PROGRAM SC_MAIN_FSM
VAR
	main_fsm	: FB_Main_FSM;
	
END_VAR

main_fsm(currentCmd := GVL_FSM.E_CommandGlobal, EmergencyReason := GVL_FSM.E_EmergencyReasonGlobal);

END_PROGRAM

(* stored: Version 1.1.0.1
   POU SC_MAIN_FSM: Id {8ae7d21a-5b8b-4fb0-8d34-ff7e9a16183c}, SpecialFunc None *)
